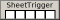
VISUALIZATION _VISU_CameraTrigger  // 60x20
VAR_IN_OUT
	mInst : FB_CameraTrigger;
END_VAR
    RoundedRectangle (0,0 60x20), tooltip "Trigger Armed", colour toggle: mInst.bTriggerArmed
    RoundedRectangle (15,10 10x10), tooltip "Speed valid", colour toggle: mInst.bSpeedValid
    RoundedRectangle (25,10 10x10), tooltip "AutomaticMode or ManualTeach", colour toggle: mInst._bCamManualTeachMode OR mInst.bI_AutomaticMode
    RoundedRectangle (35,10 10x10), tooltip "Inhibit trigger", colour toggle: NOT mInst.bInhibitTrigger
    RoundedRectangle (45,10 10x10), tooltip "HwEnable", colour toggle: mInst.bI_HwEnable
    RoundedRectangle (5,10 10x10), tooltip "Init ok", colour toggle: mInst.bInitOk
    Rectangle (0,0 60x10), "SheetTrigger", tooltip "SheetDetect"
END_VISUALIZATION

(* stored: Version 1.1.0.1, ProductVersion 3.1.4024.11
   Visu _VISU_CameraTrigger: Id {0a8a3624-dadc-420c-a93e-aadffc477bdb} *)
